FUNCTION_BLOCK POSTGRE_DB_INSERT_1
  {SET_ATTRIBUTE(OpcUa, SERVICE)}
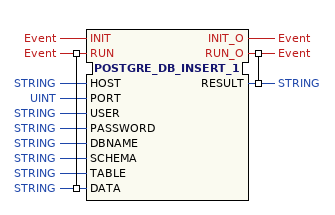
  EVENT_INPUT
    INIT;
    RUN WITH DATA, SENSOR_ID_LIST;
  END_EVENT
  EVENT_OUTPUT
    INIT_O;
    RUN_O WITH RESULT;
  END_EVENT
  VAR_INPUT
    HOST : STRING;
    PORT : UINT;
    USER : STRING;
    PASSWORD : STRING;
    DBNAME : STRING;
    SCHEMA : STRING;
    TABLE : STRING;
    DATA : STRING;
  END_VAR
  VAR_OUTPUT
    RESULT : STRING;
  END_VAR
END_FUNCTION_BLOCK
